{attribute 'GeneratedUsingTerminal: EL5001-0000-1017'}
{attribute addProperty BoxType "EL5001-0000-1017"}
{attribute addProperty Id "SSI_InputsAT %I*SSI_Inputs_0E3D8E3310WcStateAT %I*WcState_9091E0EB2InfoDataAT %I*InfoData_94A18F5E2"}
{attribute addProperty CRC "2581321518"}
{attribute addProperty Size "14"}
TYPE EL5001_99DBD72E EXTENDS EtcSlaveTerminalBase_947E5A46 :
STRUCT
	{attribute addProperty Name "SSI_Inputs"}
	SSI_Inputs : SSI_Inputs_0E3D8E33;
	{attribute addProperty Name "WcState"}
	WcState : WcState_9091E0EB;
	{attribute addProperty Name "InfoData"}
	InfoData : InfoData_94A18F5E;
END_STRUCT
END_TYPE

(* stored: Version 1.2.0.0, ProductVersion 3.1.4024.9
   DUT EL5001_99DBD72E: Id {1fab0c17-0ba7-4712-ade3-bbe845b39491} *)
